(* IEC 61131-3 sources: repolevel_ST_code_completion/output/full_case_fixed/repoeval_PID_controller/readful_result_history, 12 files *)

(* ---- HeatExchanger2_0.st ---- *)
// AJ Jaworowski 2015-02-23
// Following the presentation on
// http://openenergymonitor.org/emon/node/2999
FUNCTION_BLOCK HeatExchanger2
VAR_INPUT
	Heat_In:		REAL;		//In principle a radiator in the room [W]
	U:				REAL;		//Thermal conductance [W/K]
	TC:				REAL;		//Thermal capacity [J/K], commonly cv, specific heat capacity [J/kgK]
								//we use a smaller value than in reality, so that we can see changes
								//during a life-time...
	Temp_In:		REAL;		//Start temperature in the room [K]
	Temp_Out:		REAL;		//Outside temperature [K]
	Sample_time:	TIME;
END_VAR
VAR_OUTPUT
	Temp:			REAL;		//The resulting room temperature
END_VAR
VAR
	now: TIME;
	lastTime: TIME := T#0s;
	delta_t: REAL;
	heat_flow: REAL;
	lastTemp: REAL;
END_VAR
VAR CONSTANT
	millis: REAL := 1000;
END_VAR

now := TIME();
IF ((now - lastTime) > Sample_time) THEN
	delta_t := REAL_TO_TIME((now - lastTime)) / millis;
	heat_flow := Heat_In + U * (Temp_Out - Temp_In);
	Temp := Temp_In + (heat_flow / TC) * delta_t;
	lastTime := now;
END_IF;
END_FUNCTION_BLOCK

(* ---- HeatExchanger2_1.st ---- *)
// AJ Jaworowski 2015-02-23
// Following the presentation on
// http://openenergymonitor.org/emon/node/2999
FUNCTION_BLOCK HeatExchanger2
VAR_INPUT
	Heat_In:		REAL;		//In principle a radiator in the room [W]
	U:				REAL;		//Thermal conductance [W/K]
	TC:				REAL;		//Thermal capacity [J/K], commonly cv, specific heat capacity [J/kgK]
								//we use a smaller value than in reality, so that we can see changes
								//during a life-time...
	Temp_In:		REAL;		//Start temperature in the room [K]
	Temp_Out:		REAL;		//Outside temperature [K]
	Sample_time:	TIME;
END_VAR
VAR_OUTPUT
	Temp:			REAL;		//The resulting room temperature
END_VAR
VAR
	now: TIME;
	lastTime: TIME := T#0s;
	delta_t: REAL;
	heat_flow: REAL;
	lastTemp: REAL;
END_VAR
VAR CONSTANT
	millis: REAL := 1000;
END_VAR

now := SysTimeRtc.SysTimeGetms(); // Use SysTimeRtc library to get time in milliseconds
IF ((now - lastTime) > TO_LREAL(Sample_time)) THEN // Convert Sample_time to LREAL for comparison
  delta_t := LREAL_TO_REAL(TO_LREAL(now - lastTime) / millis);  // Ensure all arithmetic is consistent
  heat_flow := Heat_In + U * (Temp_Out - Temp_In);
  Temp := Temp_In + (heat_flow / TC) * delta_t;
  lastTime := now;
END_IF;
END_FUNCTION_BLOCK

(* ---- HeatExchanger2_2.st ---- *)
// AJ Jaworowski 2015-02-23
// Following the presentation on
// http://openenergymonitor.org/emon/node/2999
FUNCTION_BLOCK HeatExchanger2
VAR_INPUT
	Heat_In:		REAL;		//In principle a radiator in the room [W]
	U:				REAL;		//Thermal conductance [W/K]
	TC:				REAL;		//Thermal capacity [J/K], commonly cv, specific heat capacity [J/kgK]
								//we use a smaller value than in reality, so that we can see changes
								//during a life-time...
	Temp_In:		REAL;		//Start temperature in the room [K]
	Temp_Out:		REAL;		//Outside temperature [K]
	Sample_time:	TIME;
END_VAR
VAR_OUTPUT
	Temp:			REAL;		//The resulting room temperature
END_VAR
VAR
	now: TIME;
	lastTime: TIME := T#0s;
	delta_t: REAL;
	heat_flow: REAL;
	lastTemp: REAL;
END_VAR
VAR CONSTANT
	millis: REAL := 1000;
END_VAR

now := TIME(); // Assign current time (no explicit external library function needed)
IF ((now - lastTime) > Sample_time) THEN // Compare time difference with Sample_time directly
 delta_t := REAL_TO_TIME(now - lastTime) / millis; // Convert time difference to seconds (REAL format)
 heat_flow := Heat_In + U * (Temp_Out - Temp_In);
 Temp := Temp_In + (heat_flow / TC) * delta_t;
 lastTime := now;
END_IF;
END_FUNCTION_BLOCK

(* ---- HeatExchanger2_3.st ---- *)
// AJ Jaworowski 2015-02-23
// Following the presentation on
// http://openenergymonitor.org/emon/node/2999
FUNCTION_BLOCK HeatExchanger2
VAR_INPUT
	Heat_In:		REAL;		//In principle a radiator in the room [W]
	U:				REAL;		//Thermal conductance [W/K]
	TC:				REAL;		//Thermal capacity [J/K], commonly cv, specific heat capacity [J/kgK]
								//we use a smaller value than in reality, so that we can see changes
								//during a life-time...
	Temp_In:		REAL;		//Start temperature in the room [K]
	Temp_Out:		REAL;		//Outside temperature [K]
	Sample_time:	TIME;
END_VAR
VAR_OUTPUT
	Temp:			REAL;		//The resulting room temperature
END_VAR
VAR
	now: TIME;
	lastTime: TIME := T#0s;
	delta_t: REAL;
	heat_flow: REAL;
	lastTemp: REAL;
END_VAR
VAR CONSTANT
	millis: REAL := 1000;
END_VAR

now := lastTime + Sample_time; // Update 'now' using lastTime and Sample_time, simulating elapsed time
IF ((now - lastTime) > Sample_time) THEN // Compare time difference with Sample_time directly
delta_t := TO_REAL((now - lastTime)) / millis; // Convert time difference to seconds (REAL format)
heat_flow := Heat_In + U * (Temp_Out - Temp_In);
Temp := Temp_In + (heat_flow / TC) * delta_t;
lastTime := now; // Update lastTime with the current timestamp
END_IF;
END_FUNCTION_BLOCK

(* ---- HeatExchanger_0.st ---- *)
// AJ Jaworowski 2015-02-22
// Following the recipe by  Peter Nachtwey
// http://www.controlguru.com/wp/p80.html
FUNCTION_BLOCK HeatExchanger
VAR_INPUT
	Kp: REAL; //System gain
	Tp: REAL; //Process time
	CO: REAL; //Output from controller
	Dead_t: REAL; //The time before the system responds to the disturbance
	C: REAL; //Initial steady state value
	Sample_time: TIME;
END_VAR
VAR_OUTPUT
	PV: REAL; //Process value at t1
END_VAR
VAR
	now: TIME;
	lastTime: TIME;
	lastPV: REAL := 140;
	A: REAL;
	B: REAL;
	delta_t: REAL;
	DeadTimeElapsed: TIME := T#0ms;
	DeadTimeActive: BOOL := FALSE;
END_VAR
VAR CONSTANT
	millis: REAL := 1000;
END_VAR

now := TIME();
IF ((now - lastTime) > Sample_time) THEN
	delta_t := TIME_TO_REAL(Sample_time) / millis;
	A := EXP(-delta_t / Tp);
	B := 1 - A;

	IF DeadTimeActive THEN
		DeadTimeElapsed := DeadTimeElapsed + Sample_time;
		IF DeadTimeElapsed >= Dead_t THEN
			DeadTimeActive := FALSE;
			DeadTimeElapsed := T#0ms;
		END_IF
	END_IF

	IF NOT DeadTimeActive THEN
		PV := A * lastPV + B * Kp * CO + C;
		lastPV := PV;
		DeadTimeActive := TRUE;
	END_IF

	lastTime := now;
END_IF;
END_FUNCTION_BLOCK

(* ---- HeatExchanger_1.st ---- *)
// AJ Jaworowski 2015-02-22
// Following the recipe by  Peter Nachtwey
// http://www.controlguru.com/wp/p80.html
FUNCTION_BLOCK HeatExchanger
VAR_INPUT
	Kp: REAL; //System gain
	Tp: REAL; //Process time
	CO: REAL; //Output from controller
	Dead_t: REAL; //The time before the system responds to the disturbance
	C: REAL; //Initial steady state value
	Sample_time: TIME;
END_VAR
VAR_OUTPUT
	PV: REAL; //Process value at t1
END_VAR
VAR
	now: TIME;
	lastTime: TIME;
	lastPV: REAL := 140;
	A: REAL;
	B: REAL;
	delta_t: REAL;
	DeadTimeElapsed: TIME := T#0ms;
	DeadTimeActive: BOOL := FALSE;
END_VAR
VAR CONSTANT
	millis: REAL := 1000;
END_VAR

now := TIME(); // Replace invalid `SYSTEM` function. Use TRUE Codesys replacement like `SysTimeRtc.SysTimeGetMs()`.
IF ((now - lastTime) > Sample_time) THEN
	delta_t := TIME_TO_REAL(Sample_time) / millis;
	A := EXP(-delta_t / Tp);
	B := 1 - A;

	IF DeadTimeActive THEN
		DeadTimeElapsed := DeadTimeElapsed + Sample_time;
		IF DeadTimeElapsed >= Dead_t THEN
			DeadTimeActive := FALSE;
			DeadTimeElapsed := T#0ms;
		END_IF
	END_IF

	IF NOT DeadTimeActive THEN
		PV := A * lastPV + B * Kp * CO + C;
		lastPV := PV;
		DeadTimeActive := TRUE;
	END_IF

	lastTime := now;
END_IF;
END_FUNCTION_BLOCK

(* ---- HeatExchanger_2.st ---- *)
// AJ Jaworowski 2015-02-22
// Following the recipe by  Peter Nachtwey
// http://www.controlguru.com/wp/p80.html
FUNCTION_BLOCK HeatExchanger
VAR_INPUT
	Kp: REAL; //System gain
	Tp: REAL; //Process time
	CO: REAL; //Output from controller
	Dead_t: REAL; //The time before the system responds to the disturbance
	C: REAL; //Initial steady state value
	Sample_time: TIME;
END_VAR
VAR_OUTPUT
	PV: REAL; //Process value at t1
END_VAR
VAR
	now: TIME;
	lastTime: TIME;
	lastPV: REAL := 140;
	A: REAL;
	B: REAL;
	delta_t: REAL;
	DeadTimeElapsed: TIME := T#0ms;
	DeadTimeActive: BOOL := FALSE;
END_VAR
VAR CONSTANT
	millis: REAL := 1000;
END_VAR

now := SysTimeRtc.SysTimeGetMs(); // Replace invalid `TIME()` function with system function for elapsed time.
IF ((now - lastTime) > Sample_time) THEN
delta_t := REAL_TO_TIME(Sample_time) / millis; // Corrected conversion operation for type matching consistency.
	A := EXP(-delta_t / Tp);
	B := 1 - A;

	IF DeadTimeActive THEN
		DeadTimeElapsed := DeadTimeElapsed + Sample_time;
		IF DeadTimeElapsed >= Dead_t THEN
			DeadTimeActive := FALSE;
			DeadTimeElapsed := T#0ms;
		END_IF
	END_IF

	IF NOT DeadTimeActive THEN
		PV := A * lastPV + B * Kp * CO + C;
		lastPV := PV;
		DeadTimeActive := TRUE;
	END_IF

	lastTime := now;
END_IF;
END_FUNCTION_BLOCK

(* ---- HeatExchanger_3.st ---- *)
// AJ Jaworowski 2015-02-22
// Following the recipe by  Peter Nachtwey
// http://www.controlguru.com/wp/p80.html
FUNCTION_BLOCK HeatExchanger
VAR_INPUT
	Kp: REAL; //System gain
	Tp: REAL; //Process time
	CO: REAL; //Output from controller
	Dead_t: REAL; //The time before the system responds to the disturbance
	C: REAL; //Initial steady state value
	Sample_time: TIME;
END_VAR
VAR_OUTPUT
	PV: REAL; //Process value at t1
END_VAR
VAR
	now: TIME;
	lastTime: TIME;
	lastPV: REAL := 140;
	A: REAL;
	B: REAL;
	delta_t: REAL;
	DeadTimeElapsed: TIME := T#0ms;
	DeadTimeActive: BOOL := FALSE;
END_VAR
VAR CONSTANT
	millis: REAL := 1000;
END_VAR

now := SysTimeRtc.SysTimeGet(); // Correct system function for getting the current time in type TIME.
IF ((TIME_TO_REAL(now - lastTime) / 1000.0) > TIME_TO_REAL(Sample_time)) THEN // Convert TIME type to REAL for comparison.
delta_t := TIME_TO_REAL(Sample_time) / millis; // Correct conversion from TIME to REAL for division.
	A := EXP(-delta_t / Tp);
	B := 1 - A;

	IF DeadTimeActive THEN
		DeadTimeElapsed := DeadTimeElapsed + Sample_time;
		IF DeadTimeElapsed >= Dead_t THEN
			DeadTimeActive := FALSE;
			DeadTimeElapsed := T#0ms;
		END_IF
	END_IF

	IF NOT DeadTimeActive THEN
		PV := A * lastPV + B * Kp * CO + C;
		lastPV := PV;
		DeadTimeActive := TRUE;
	END_IF

	lastTime := now;
END_IF;
END_FUNCTION_BLOCK

(* ---- PID_controller_0.st ---- *)
//***************************************************************
//* A simple PID controller for Codesys.
//* by Alexander Jaworowski
//* Inspiration from https://github.com/br3ttb/Arduino-PID-Library
//* https://github.com/alexjaw/PID_controller
//* This Library is licensed under a MIT License
//
// 2015-02-22	Bug fix in the calculation of CO_I.
//				Added derivative term (d(err)/dt = -d(PV)/dt, i.e.
//				derivative on measurements
//***************************************************************
FUNCTION_BLOCK PID_controller
VAR_INPUT
	SP : REAL;
	PV : REAL;
	Kc : REAL;
	Ti : REAL;
	Td : REAL;
	SampleTime: TIME; //Should be ~0.1 * Tp, Tp : the process time [http://www.controlguru.com/2007/012807.html]
	LowerLimit: REAL;
	UpperLimit: REAL;
END_VAR
VAR_OUTPUT
	CO: REAL; //Controller Output
	CO_P: REAL; //Prportional term
	CO_I: REAL; //Integral term
	CO_D: REAL; //Derivative term
END_VAR
VAR CONSTANT
	millis: UINT := 1000;
END_VAR
VAR
	lastErr: REAL := 0; //Previous error
	integral: REAL := 0; //Integral accumulator
	deltaTime: REAL := 0; //Time difference in seconds
	deltaPV: REAL := 0; //Change in process variable
END_VAR

now := TIME(); //Get current time
deltaTime := REAL_TO_TIME((now - lastTime)) / millis; //Calculate elapsed time in seconds

IF deltaTime >= REAL_TO_TIME(SampleTime) THEN
	// Calculate error
	err := SP - PV;

	// Proportional term
	CO_P := Kc * err;

	// Integral term with anti-windup
	integral := integral + (err * deltaTime);
	IF integral > UpperLimit THEN
		integral := UpperLimit;
	ELSIF integral < LowerLimit THEN
		integral := LowerLimit;
	END_IF;
	CO_I := (Kc / Ti) * integral;

	// Derivative term
	deltaPV := PV - lastErr;
	CO_D := -(Kc * Td * deltaPV / deltaTime);

	// Compute total output
	CO := CO_P + CO_I + CO_D;

	// Apply output limits
	IF CO > UpperLimit THEN
		CO := UpperLimit;
	ELSIF CO < LowerLimit THEN
		CO := LowerLimit;
	END_IF;

	// Update last values
	lastErr := PV;
	lastTime := now;
END_IF;
END_FUNCTION_BLOCK

(* ---- PID_controller_1.st ---- *)
//***************************************************************
//* A simple PID controller for Codesys.
//* by Alexander Jaworowski
//* Inspiration from https://github.com/br3ttb/Arduino-PID-Library
//* https://github.com/alexjaw/PID_controller
//* This Library is licensed under a MIT License
//
// 2015-02-22	Bug fix in the calculation of CO_I.
//				Added derivative term (d(err)/dt = -d(PV)/dt, i.e.
//				derivative on measurements
//***************************************************************
FUNCTION_BLOCK PID_controller
VAR_INPUT
	SP : REAL;
	PV : REAL;
	Kc : REAL;
	Ti : REAL;
	Td : REAL;
	SampleTime: TIME; //Should be ~0.1 * Tp, Tp : the process time [http://www.controlguru.com/2007/012807.html]
	LowerLimit: REAL;
	UpperLimit: REAL;
END_VAR
VAR_OUTPUT
	CO: REAL; //Controller Output
	CO_P: REAL; //Prportional term
	CO_I: REAL; //Integral term
	CO_D: REAL; //Derivative term
END_VAR
VAR CONSTANT
	millis: UINT := 1000;
END_VAR
VAR
	lastErr: REAL := 0; //Previous error
	integral: REAL := 0; //Integral accumulator
	deltaTime: REAL := 0; //Time difference in seconds
	deltaPV: REAL := 0; //Change in process variable
END_VAR

// Declare "now" and "lastTime" under VAR and fix calculation
  now := TIME(); // Get current time
  deltaTime := TO_REAL(now - lastTime) / TO_REAL(T#1S); // Calculate elapsed time in seconds

IF deltaTime >= REAL_TO_TIME(SampleTime) THEN
	// Calculate error
	err := SP - PV;

	// Proportional term
	CO_P := Kc * err;

	// Integral term with anti-windup
	integral := integral + (err * deltaTime);
	IF integral > UpperLimit THEN
		integral := UpperLimit;
	ELSIF integral < LowerLimit THEN
		integral := LowerLimit;
	END_IF;
	CO_I := (Kc / Ti) * integral;

	// Derivative term
	deltaPV := PV - lastErr;
	CO_D := -(Kc * Td * deltaPV / deltaTime);

	// Compute total output
	CO := CO_P + CO_I + CO_D;

	// Apply output limits
	IF CO > UpperLimit THEN
		CO := UpperLimit;
	ELSIF CO < LowerLimit THEN
		CO := LowerLimit;
	END_IF;

	// Update last values
	lastErr := PV;
	lastTime := now;
END_IF;
END_FUNCTION_BLOCK

(* ---- Tank_0.st ---- *)
//A.J. Jaworowski 2015-02-20
//Simulering av en tank med RedBull
FUNCTION_BLOCK Tank
VAR_INPUT
	Process_In: REAL;  //Flöde in per sekund, testa vad som händer on du matar in 100
					   //Därefter ska regulatorns OUT in i denna ingång.
	Process_Out: REAL; //Flöde ut per sekund, typ 90
					   //Effekten blir att tanken fylls med 10 per sekund
					   //Full efter ca 1 minut - testa
	SampleTime: TIME;  //Uppdateringstid, typ 100ms
	Lower_limit: REAL; //Tankens lägsta nivå, typ 0
	Upper_limit: REAL; //Tankens max nivå, kanske 500
END_VAR
VAR_OUTPUT
	Level: REAL; //Nivån i tanken
END_VAR
VAR
	now: TIME;
	lastTime: TIME := T#0ms;
	millis: UINT := 1000;
	temp: REAL;
END_VAR

now := TIME();
IF (now - lastTime) >= SampleTime THEN
	temp := TIME_TO_REAL(SampleTime) / millis * (Process_In - Process_Out);
	Level := Level + temp;

	IF Level < Lower_limit THEN
		Level := Lower_limit;
	ELSIF Level > Upper_limit THEN
		Level := Upper_limit;
	END_IF;

	lastTime := now;
END_IF;
END_FUNCTION_BLOCK

(* ---- Tank_2.st ---- *)
//A.J. Jaworowski 2015-02-20
//Simulering av en tank med RedBull
FUNCTION_BLOCK Tank
VAR_INPUT
	Process_In: REAL;  //Flöde in per sekund, testa vad som händer on du matar in 100
					   //Därefter ska regulatorns OUT in i denna ingång.
	Process_Out: REAL; //Flöde ut per sekund, typ 90
					   //Effekten blir att tanken fylls med 10 per sekund
					   //Full efter ca 1 minut - testa
	SampleTime: TIME;  //Uppdateringstid, typ 100ms
	Lower_limit: REAL; //Tankens lägsta nivå, typ 0
	Upper_limit: REAL; //Tankens max nivå, kanske 500
END_VAR
VAR_OUTPUT
	Level: REAL; //Nivån i tanken
END_VAR
VAR
	now: TIME;
	lastTime: TIME := T#0ms;
	millis: UINT := 1000;
	temp: REAL;
END_VAR

now := lastTime + SampleTime; // Simulating a time increment based on SampleTime
IF (now - lastTime) >= SampleTime THEN
  temp := REAL(toDINT(SampleTime) / toDINT(T#1ms)) / millis * (Process_In - Process_Out); // Converting TIME to REAL
  Level := Level + temp;

  IF Level < Lower_limit THEN
    Level := Lower_limit;
  ELSIF Level > Upper_limit THEN
    Level := Upper_limit;
  END_IF;

  lastTime := now; // Update lastTime to the current simulated time
END_IF;
END_FUNCTION_BLOCK
